// TIA Portal V20 export
// export: Created 2025-12-01T14:57:27.8084836Z, ExportSetting None, DisplayName Totally Integrated Automation Portal, DisplayVersion V20 Update 3, DisplayName TIA Portal Openness, DisplayVersion V20 Update 3, DisplayName TIA Portal Version Control Interface, DisplayVersion V20 Update 3, DisplayName STEP 7 Professional, DisplayVersion V20 Update 3, DisplayName STEP 7 Safety, DisplayVersion V20 Update 2, DisplayName WinCC Basic/Comfort/Advanced, DisplayVersion V20 Update 3, DisplayName WinCC Professional, DisplayVersion V20 Update 3, DisplayName WinCC Unified, DisplayVersion V20 Update 3
FUNCTION_BLOCK "FB603_EntradaMovil_Frontal_Quimarox"   // FB603, LAD
{ S7_Optimized_Access := 'FALSE' }
// stored: AutoNumber false, SetENOAutomatically false
   VAR_INPUT
      MesaDeCarga : UInt;
      ID_Quimarox : UInt;
      ID_Elemento : UInt;
      EnTension : Bool;
      Termico_Tilt : Bool;
      pHs_PosicionCarga : Bool;
      pHs_Protrusion : Bool;
      En_PosicionReposo : Bool;
      Corte_PosicionReposo : Bool;
      Corte_PosicionCarga : Bool;
      En_PosicionCarga : Bool;
      PRV_AVTF : Bool;
      PRV_DescargaActiva : Bool;
      V_FILTRO_pHsPresencia : Int;
      Pto_Ajuste_1 : Int;
      Pto_Ajuste_2 : Int;
      Pto_Ajuste_3 : Int;
      Pto_Ajuste_4 : Int;
      Pto_Ajuste_5 : Int;
      Pto_Ajuste_6 : Int;
   END_VAR
   VAR_OUTPUT
      Permiso_DeCarga : Bool;
      PararElevador : Bool;
      ElevadorEnLenta : Bool;
      AvanceCorreas : Bool;
      Ir_PosicionReposo : Bool;
      Ir_PosicionCarga : Bool;
   END_VAR
   VAR_IN_OUT
      ROUTING_Destino : UInt;
      ROUTING_Etiqueta : UDInt;
   END_VAR
   VAR
      TMP_EnTension { S7_SetPoint := 'True'} : "FB910_CNT_UHS";
      FILTRO_pHsPresencia { S7_SetPoint := 'True'} : "FB910_CNT_UHS";
      EstadoAsociadoEnMesa : UInt;
      Aux_PeineDeCarga : UInt;
   END_VAR
   VAR_TEMP
      MesaQuimarox : UInt;
      PeineReservado : UInt;
      TMP_PeineLiberar : UInt;
      NumeroUT : UInt;
      EsMesaTL : Bool;
      FILTRO_PosicionCarga : Bool;
   END_VAR
BEGIN

NETWORK
TITLE = ERROR - Rearme
/////////////////////////////////////////////////////////////
/////////////////////////////////////////////////////////////
/////////////////////////////////////////////////////////////
// Rearne de Errores
      SET;
      A     "DB902_Estado_ZonaMesa".EstadoMesas[#MesaDeCarga].Rearme_CBx;
      O     "DB902_Estado_ZonaMesa".EstadoMesas[#MesaDeCarga].PerReset_CBx;
      R     "DB900_Estado_Mesas".EstadoVI[#MesaDeCarga].Error_Mx;
      R     "DB900_Estado_Mesas".EstadoVI[#MesaDeCarga].Err_Protusion;
      R     "DB900_Estado_Mesas".EstadoVI[#MesaDeCarga].Err_TOut_Avance_E1_E3;
      R     "DB900_Estado_Mesas".EstadoVI[#MesaDeCarga].Err_Tout_Sacar;
      R     "DB900_Estado_Mesas".EstadoVI[#MesaDeCarga].Err_Tout_Recoger;
      R     "DB900_Estado_Mesas".EstadoVI[#MesaDeCarga].Err_DatosPLC;
      R     "DB900_Estado_Mesas".EstadoVI[#MesaDeCarga].Err_Termico_E2_E4;



NETWORK
TITLE = HMI - Manual
/////////////////////////////////////////////////////////////
/////////////////////////////////////////////////////////////
/////////////////////////////////////////////////////////////
// Para HMI >>> Manual
      SET;
      O     "DB902_Estado_ZonaMesa".EstadoMesas[#MesaDeCarga].Manual_CBx;
      =     "DB900_Estado_Mesas".EstadoVI[#MesaDeCarga].Manual;



NETWORK
TITLE = HMI - Entradas y Salidas de la Mesa
/////////////////////////////////////////////////////////////
/////////////////////////////////////////////////////////////
/////////////////////////////////////////////////////////////
// Entradas
      SET;
      A     #pHs_PosicionCarga;
      =     "DB900_Estado_Mesas".EstadoVI[#MesaDeCarga].En_PHS_1;
      SET;
      A     #pHs_Protrusion;
      =     "DB900_Estado_Mesas".EstadoVI[#MesaDeCarga].En_pHs_Prot1;

      SET;  // Solo el TILT
      A     #Termico_Tilt;
      =     "DB900_Estado_Mesas".EstadoVI[#MesaDeCarga].En_Termico2;

      SET;
      A     #En_PosicionReposo;
      =     "DB904_Estado_Maquinas".EstadoVI[#MesaDeCarga].Byte8_bit4;
      SET;
      A     #Corte_PosicionReposo;
      =     "DB904_Estado_Maquinas".EstadoVI[#MesaDeCarga].Byte7_bit6;
      SET;
      A     #Corte_PosicionCarga;
      =     "DB904_Estado_Maquinas".EstadoVI[#MesaDeCarga].Byte7_bit7;
      SET;
      A     #En_PosicionCarga;
      =     "DB904_Estado_Maquinas".EstadoVI[#MesaDeCarga].Byte8_bit5;


// Salidas
      SET;
      A     #Permiso_DeCarga;
      =     "DB900_Estado_Mesas".EstadoVI[#MesaDeCarga].Sa_Extender_Empujador;
      SET;
      A     #Ir_PosicionReposo;
      =     "DB900_Estado_Mesas".EstadoVI[#MesaDeCarga].Sa_Trans_Baj;
      SET;
      A     #Ir_PosicionCarga;
      =     "DB900_Estado_Mesas".EstadoVI[#MesaDeCarga].Sa_Trans_Sub;



NETWORK
TITLE = Comprobacion de que la MESA es de TRACKING
/////////////////////////////////////////////////////////////////////////////////////
/////////////////////////////////////////////////////////////////////////////////////
/////////////////////////////////////////////////////////////////////////////////////
// Comprobar si es una Mesa de Tracking o Routing
      SET;
      A     "DB850_DefinicionMesas".Mesa[#MesaDeCarga].ConfigMesa.MesaTL;
      =     #EsMesaTL;



REGION Network 5: TMP - Espera En Tension
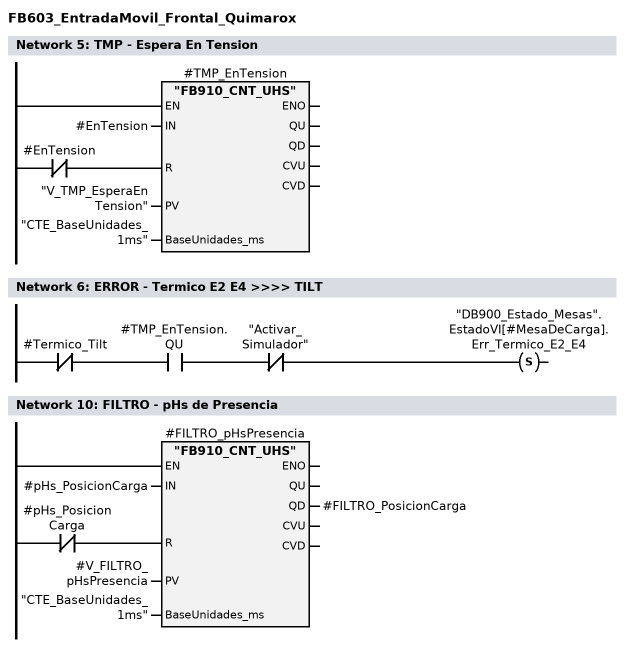
   RUNG wire#powerrail
      #TMP_EnTension(R := wire#w1, IN := #EnTension, PV := "V_TMP_EsperaEnTension", BaseUnidades_ms := "CTE_BaseUnidades_1ms", QU =>, QD =>, CVU =>, CVD =>)
   END_RUNG
   RUNG wire#powerrail
      I_Contact( #EnTension )
   END_RUNG wire#w1
   // the same network as SCL:
   #TMP_EnTension(IN := #EnTension,   // "FB910_CNT_UHS"
                  R := NOT #EnTension,
                  PV := "V_TMP_EsperaEnTension",
                  BaseUnidades_ms := "CTE_BaseUnidades_1ms");
END_REGION

REGION Network 6: ERROR - Termico E2 E4 >>>> TILT
   RUNG wire#powerrail
      I_Contact( #Termico_Tilt )
      Contact( #TMP_EnTension.QU )
      I_Contact( "Activar_Simulador" )
      S_Coil( "DB900_Estado_Mesas".EstadoVI[#MesaDeCarga].Err_Termico_E2_E4 )
   END_RUNG
   // the same network as SCL:
   IF NOT #Termico_Tilt AND #TMP_EnTension.QU AND NOT "Activar_Simulador" THEN
       "DB900_Estado_Mesas".EstadoVI[#MesaDeCarga].Err_Termico_E2_E4 := TRUE;
   END_IF;
END_REGION

NETWORK
TITLE = INICIALIZACION - Previa
/////////////////////////////////////////////////////////////////////////////////////
/////////////////////////////////////////////////////////////////////////////////////
/////////////////////////////////////////////////////////////////////////////////////
      CLR;
      =     #PararElevador;
      =     #ElevadorEnLenta;

      CLR;
      =     #Permiso_DeCarga;

      CLR;
      =     #AvanceCorreas;
      =     #Ir_PosicionReposo;
      =     #Ir_PosicionCarga;



NETWORK
TITLE = SISTEMA - Reset
/////////////////////////////////////////////////////////////
/////////////////////////////////////////////////////////////
/////////////////////////////////////////////////////////////
// - Existe RESET ??
      SET;
      AN    "DB902_Estado_ZonaMesa".EstadoMesas[#MesaDeCarga].PerReset_CBx;  //#Estado_CBx.PerReset_CBx
      JC    NoRealizandose_Reset;

      L     0;
      T     #EstadoAsociadoEnMesa;


/////////////////////////////////////////////////////////////
/////////////////////////////////////////////////////////////
/////////////////////////////////////////////////////////////
// - Final Tratamiento del RESET
NoRealizandose_Reset:NOP   0;



NETWORK
TITLE = >>>>>>>>>>>>>>>>>>>>>>>>>>>>>>>>>>>>>>>>>>>>>>>>>>>>>>>>>>>>>>>>>>>

REGION Network 10: FILTRO - pHs de Presencia
   RUNG wire#powerrail
      #FILTRO_pHsPresencia(R := wire#w1, IN := #pHs_PosicionCarga, PV := #V_FILTRO_pHsPresencia, BaseUnidades_ms := "CTE_BaseUnidades_1ms", QU =>, QD => #FILTRO_PosicionCarga, CVU =>, CVD =>)
   END_RUNG
   RUNG wire#powerrail
      I_Contact( #pHs_PosicionCarga )
   END_RUNG wire#w1
   // the same network as SCL:
   #FILTRO_pHsPresencia(IN := #pHs_PosicionCarga,   // "FB910_CNT_UHS"
                        R := NOT #pHs_PosicionCarga,
                        PV := #V_FILTRO_pHsPresencia,
                        BaseUnidades_ms := "CTE_BaseUnidades_1ms",
                        QD => #FILTRO_PosicionCarga);
END_REGION

NETWORK
TITLE = >>>>>>>>>>>>>>>>>>>>>>>>>>>>>>>>>>>>>>>>>>>>>>>>>>>>>>>>>>>>>>>>>>>

NETWORK
TITLE = Disrtibucion >>> Control Etapa Activa
/////////////////////////////////////////////////////////////////////////////////////
/////////////////////////////////////////////////////////////////////////////////////
/////////////////////////////////////////////////////////////////////////////////////
// listado de saltos de programa
      L     #EstadoAsociadoEnMesa;
      JL    ESTADO_PorDefecto;

      JU    ETAPA_00_EnReset;
      JU    ETAPA_01_EnReposo;

      JU    ETAPA_02_PrevioCarga_ComprobarRuta;
      JU    ETAPA_03_PrevioCarga_ReservaPeine;
      JU    ETAPA_04_PrevioCarga_Sincroniza;
      JU    ETAPA_05_PrevioCarga_MoverPosicionDeCarga;
      JU    ETAPA_06_CargaDelPeine;
      JU    ETAPA_07_FinCargaDelPeine;
      JU    ETAPA_08_VolverReposo;

      JU    ESTADO_PorDefecto;

      JU    ETAPA_10_ResetCargado_ComprobarRuta;
      JU    ETAPA_11_ResetVacio_MoverPosicionDeReposo;

ESTADO_PorDefecto:JU    FinFuncion;



NETWORK
TITLE = ETAPA 00 >>> Etapa Reset >>>> PENDIENTE
/////////////////////////////////////////////////////////////////////////////////////
/////////////////////////////////////////////////////////////////////////////////////
/////////////////////////////////////////////////////////////////////////////////////
ETAPA_00_EnReset:NOP   0;
      SET;
      =     "DB900_Estado_Mesas".EstadoVI[#MesaDeCarga].Etapas_Reset;

/////////////////////////////////////////////////////////////////////////////////////
// error de protusion
      SET;
      AN    #pHs_Protrusion;
      JC    ErrorProtrusion;


/////////////////////////////////////////////////////////////////////////////////////
// Tiene que estar en Marcha y Sin Error para continuar
      SET;
      AN    "DB902_Estado_ZonaMesa".EstadoMesas[#MesaDeCarga].Marcha_CBx;
      O     "DB902_Estado_ZonaMesa".EstadoMesas[#MesaDeCarga].Error_CBx;
      JC    ET00_PararElevador;



/////////////////////////////////////////////////////////////////////////////////////
// En Resposo
      SET;
      A     #En_PosicionReposo;
      JC    ET00_IrEtapa_01_EnReposo;

/////////////////////////////////////////////////////////////////////////////////////
// NO Reposo - Vacio
      SET;
      AN    #FILTRO_PosicionCarga;
      JC    ET00_IrEtapa_11_ResetVacio_MoverPosicionReposo;

/////////////////////////////////////////////////////////////////////////////////////
// NO Reposo - Con Carga
      SET;
      A     #FILTRO_PosicionCarga;
      JC    ET00_IrEtapa_10_ResetCargado_ComprobarRuta;


/////////////////////////////////////////////////////////////////////////////////////
// Final del Reparto  ?????? No DEBE LLEGAR AQUI
      BE;


/////////////////////////////////////////////////////////////////////////////////////
/////////////////////////////////////////////////////////////////////////////////////
/////////////////////////////////////////////////////////////////////////////////////
ET00_PararElevador:NOP   0;
      SET;
      =     #PararElevador;
      BE;


/////////////////////////////////////////////////////////////////////////////////////
/////////////////////////////////////////////////////////////////////////////////////
/////////////////////////////////////////////////////////////////////////////////////
ET00_IrEtapa_01_EnReposo:NOP   0;
      L     1;
      T     #EstadoAsociadoEnMesa;
      JU    ETAPA_01_EnReposo;

/////////////////////////////////////////////////////////////////////////////////////
ET00_IrEtapa_10_ResetCargado_ComprobarRuta:NOP   0;
      L     10;
      T     #EstadoAsociadoEnMesa;
      JU    ETAPA_10_ResetCargado_ComprobarRuta;

/////////////////////////////////////////////////////////////////////////////////////
ET00_IrEtapa_11_ResetVacio_MoverPosicionReposo:NOP   0;
      L     11;
      T     #EstadoAsociadoEnMesa;
      JU    ETAPA_11_ResetVacio_MoverPosicionDeReposo;



NETWORK
TITLE = ETAPA 01 >>> Etapa Reposo >>> Esta Vacia
/////////////////////////////////////////////////////////////////////////////////////
/////////////////////////////////////////////////////////////////////////////////////
/////////////////////////////////////////////////////////////////////////////////////
// estado reposo
ETAPA_01_EnReposo:NOP   0;
      SET;
      =     "DB900_Estado_Mesas".EstadoVI[#MesaDeCarga].Etapa_Vacia;


/////////////////////////////////////////////////////////////////////////////////////
// error de protusion
      SET;
      AN    #pHs_Protrusion;
      JC    ErrorProtrusion;

/////////////////////////////////////////////////////////////////////////////////////
/////////////////////////////////////////////////////////////////////////////////////
/////////////////////////////////////////////////////////////////////////////////////
// Si Viene un Peine >>> Reservado para el Elemento >>> LIBERAR Peine
      SET;  // --- Sin Ventana
      AN    "DB602_ElementosQuimarox".Quimarox[#ID_Quimarox].Elementos[#ID_Elemento].Hay_Carrier_en_ventana;
      JC    ET01_PorReserva_NoLiberarPeine;

      L     "DB602_ElementosQuimarox".Quimarox[#ID_Quimarox].Elementos[#ID_Elemento].Numero_carrier;
      T     #TMP_PeineLiberar;

      SET;  // --- Sin Reserva
      AN    "DB601_PeinesQuimarox".Quimarox[#ID_Quimarox].vagon[#TMP_PeineLiberar].vagon_reservado_carga;
      JC    ET01_PorReserva_NoLiberarPeine;

      SET;  // --- No es para el elemento
      L     "DB601_PeinesQuimarox".Quimarox[#ID_Quimarox].vagon[#TMP_PeineLiberar].punto_entrada_carga;
      L     #ID_Elemento;
      <>I;
      JC    ET01_PorReserva_NoLiberarPeine;

/////////////////////////////////////////////////////////////////////////////////////
      SET;  // --- Liberar Peine
      R     "DB601_PeinesQuimarox".Quimarox[#ID_Quimarox].vagon[#TMP_PeineLiberar].vagon_reservado_carga;

      L     0;
      T     "DB601_PeinesQuimarox".Quimarox[#ID_Quimarox].vagon[#TMP_PeineLiberar].punto_entrada_carga;

/////////////////////////////////////////////////////////////////////////////////////
ET01_PorReserva_NoLiberarPeine:NOP   0;


/////////////////////////////////////////////////////////////////////////////////////
/////////////////////////////////////////////////////////////////////////////////////
/////////////////////////////////////////////////////////////////////////////////////
// Esta poscionado Correctamente
      SET;
      AN    #PRV_AVTF;
      AN    #FILTRO_PosicionCarga;
      A     #pHs_Protrusion;
      AN    #En_PosicionReposo;
      JC    ET01_IrEtapa_08_VolverReposo;

/////////////////////////////////////////////////////////////////////////////////////
      SET;
      AN    #PRV_AVTF;
      AN    #FILTRO_PosicionCarga;
      A     #pHs_Protrusion;
      JC    FinFuncion;

/////////////////////////////////////////////////////////////////////////////////////
      SET;
      A     #PRV_AVTF;
      AN    #FILTRO_PosicionCarga;
      A     #pHs_Protrusion;
      JC    ET01_IrEtapa_02_PrevioCarga_ComprobarRuta;

      BE;


/////////////////////////////////////////////////////////////////////////////////////
ET01_IrEtapa_08_VolverReposo:NOP   0;
      L     8;
      T     #EstadoAsociadoEnMesa;
      JU    ETAPA_08_VolverReposo;

/////////////////////////////////////////////////////////////////////////////////////
ET01_IrEtapa_02_PrevioCarga_ComprobarRuta:NOP   0;
      L     2;
      T     #EstadoAsociadoEnMesa;
      JU    ETAPA_02_PrevioCarga_ComprobarRuta;



NETWORK
TITLE = ETAPA 02 >>> Comprobar Ruta >>>>> OJO!!!!!!!!!!!!!!!
/////////////////////////////////////////////////////////////////////////////////////
// estado preparar carga
ETAPA_02_PrevioCarga_ComprobarRuta:NOP   0;
      SET;
      =     "DB900_Estado_Mesas".EstadoVI[#MesaDeCarga].Etapa_Vacia;

/////////////////////////////////////////////////////////////////////////////////////
// Error de Protrusion
      SET;
      AN    #pHs_Protrusion;
      JC    ErrorProtrusion;

/////////////////////////////////////////////////////////////////////////////////////
/// --- Comprobacion del TIPO de MESA
      SET;
      AN    #EsMesaTL;
      JC    TRACKING_ComprobarRuta;
      JU    ROUTING_ComprobarRuta;

/////////////////////////////////////////////////////////////////////////////////////
/////////////////////////////////////////////////////////////////////////////////////
/////////////////////////////////////////////////////////////////////////////////////
/// --- Comprobacion de Ruta en una MESA de ROUTING
ROUTING_ComprobarRuta:NOP   0;
      L     #ROUTING_Destino;
      L     0;
      ==I;
      JC    FinFuncion;
      JU    FINAL_ComprobacionDeRuta;

/////////////////////////////////////////////////////////////////////////////////////
/////////////////////////////////////////////////////////////////////////////////////
/////////////////////////////////////////////////////////////////////////////////////
/// --- Comprobacion de Ruta en una MESA de TRACKING
TRACKING_ComprobarRuta:NOP   0;
      L     "DB810_ColasMesas".Colas[#MesaDeCarga].UT_PrimeraMesa;
      T     #NumeroUT;

      SET;
      L     #NumeroUT;  // Debe existir UT
      L     0;
      ==I;
      JC    FinFuncion;

// si la mesa actual es la de destino, es que aun no tiene ruta, y tenemos que esperar
      SET;
      L     "DB812_UTs_Control".UT[#NumeroUT].MesaActual;
      L     "DB812_UTs_Control".UT[#NumeroUT].MesaDestino;
      ==I;
      JC    FinFuncion;

      SET;
      L     0;
      L     "DB812_UTs_Control".UT[#NumeroUT].MesaDestino;
      ==I;
      JC    FinFuncion;

      JU    FINAL_ComprobacionDeRuta;

/////////////////////////////////////////////////////////////////////////////////////
/////////////////////////////////////////////////////////////////////////////////////
/////////////////////////////////////////////////////////////////////////////////////
/// --- Final de la Comprobacion de Ruta
//      si tenemos destino, pasamos a reservar peine de carga
FINAL_ComprobacionDeRuta:NOP   0;
      L     3;
      T     #EstadoAsociadoEnMesa;
      JU    ETAPA_03_PrevioCarga_ReservaPeine;  // si ya hemos extraido la orden, pasamos a extraer el destino



NETWORK
TITLE = ETAPA 03 >>> Reserva Peine
/////////////////////////////////////////////////////////////////////////////////////
/////////////////////////////////////////////////////////////////////////////////////
/////////////////////////////////////////////////////////////////////////////////////
// extracción destino y reserva de peine
ETAPA_03_PrevioCarga_ReservaPeine:NOP   0;
      SET;
      =     "DB900_Estado_Mesas".EstadoVI[#MesaDeCarga].Etapa_Vacia;


/////////////////////////////////////////////////////////////////////////////////////
      SET;
      AN    #pHs_Protrusion;
      JC    ErrorProtrusion;

/////////////////////////////////////////////////////////////////////////////////////
// rearme del error si ha desaparecido la caja   OJO!!!!!!!CAMBIADO
      SET;
      AN    #PRV_AVTF;
      AN    #FILTRO_PosicionCarga;
      A     #pHs_Protrusion;
      A     "DB902_Estado_ZonaMesa".EstadoMesas[#MesaDeCarga].Rearme_CBx;
      JC    ET03_IrEtapa_01_EnReposo;


/////////////////////////////////////////////////////////////////////////////////////
/////////////////////////////////////////////////////////////////////////////////////
/////////////////////////////////////////////////////////////////////////////////////
// reserva de peine >>> Mesa Movil Frontal (3)
      CALL  "FC602_ReservaPeine"
      ( ID_Quimarox          := #ID_Quimarox,
        ID_ElementoPeticion  := #ID_Elemento,
        TipoDeElemento       := 3,
        NumeroPeineReservado := #PeineReservado
      );

      SET;
      L     #PeineReservado;
      L     0;
      ==I;
      JC    FinFuncion;

/////////////////////////////////////////////////////////////////////////////////////
/////////////////////////////////////////////////////////////////////////////////////
/////////////////////////////////////////////////////////////////////////////////////
      L     #PeineReservado;  // recogemos la peticion
      T     #Aux_PeineDeCarga;

      L     4;
      T     #EstadoAsociadoEnMesa;
      JU    ETAPA_04_PrevioCarga_Sincroniza;


/////////////////////////////////////////////////////////////////////////////////////
ET03_IrEtapa_01_EnReposo:NOP   0;
      L     1;
      T     #EstadoAsociadoEnMesa;
      JU    ETAPA_01_EnReposo;



NETWORK
TITLE = ETAPA 04 >>> Sincronizacion
/////////////////////////////////////////////////////////////////////////////////////
/////////////////////////////////////////////////////////////////////////////////////
/////////////////////////////////////////////////////////////////////////////////////
// a la espera de la sincronización con el peine reservado para nosotros
ETAPA_04_PrevioCarga_Sincroniza:NOP   0;
      SET;
      =     "DB900_Estado_Mesas".EstadoVI[#MesaDeCarga].Etapas_Carga_E1;


/////////////////////////////////////////////////////////////////////////////////////
// Error de Protrusion
      SET;
      AN    #pHs_Protrusion;
      JC    ErrorProtrusion;

/////////////////////////////////////////////////////////////////////////////////////
// ahora que ya estamos los datos de nuestro elemento comprobamos lo siguiente
// que tenemos delante el carrier que tenemos reservado para la carga
// que el carrier reservado para la carga está en ventana
      SET;
      A     "DB602_ElementosQuimarox".Quimarox[#ID_Quimarox].Elementos[#ID_Elemento].Hay_Carrier_en_ventana;
      A(;
      L     "DB602_ElementosQuimarox".Quimarox[#ID_Quimarox].Elementos[#ID_Elemento].Numero_carrier;  //#datos_elemento.Numero_carrier
      L     #Aux_PeineDeCarga;
      ==I;
      );
      JC    ET04_IrEtapa_05_MoverPosicionDeCarga;

      BE;

/////////////////////////////////////////////////////////////////////////////////////
ET04_IrEtapa_05_MoverPosicionDeCarga:NOP   0;
      L     5;  // saltamos al inicio de posicionamiento para carga
      T     #EstadoAsociadoEnMesa;
      JU    ETAPA_05_PrevioCarga_MoverPosicionDeCarga;



NETWORK
TITLE = ETAPA 05 >>> Mover Posicion de Carga
/////////////////////////////////////////////////////////////////////////////////////
/////////////////////////////////////////////////////////////////////////////////////
/////////////////////////////////////////////////////////////////////////////////////
ETAPA_05_PrevioCarga_MoverPosicionDeCarga:NOP   0;
      SET;
      =     "DB900_Estado_Mesas".EstadoVI[#MesaDeCarga].Etapas_Carga_E1;


      SET;
      A     #En_PosicionCarga;
      JC    ET05_IrEtapa_06_CargaDelPeine;

      SET;
      =     #Ir_PosicionCarga;
      =     #AvanceCorreas;
      =     #Permiso_DeCarga;
      CLR;
      =     #Ir_PosicionReposo;


/////////////////////////////////////////////////////////////////////////////////////
// como estamos metiendo el transportador, tenemos que vigilar que no tarda demasiado en entrar
      L     "DB602_ElementosQuimarox".Quimarox[#ID_Quimarox].Elementos[#ID_Elemento].Avance_carrier;
      L     #Pto_Ajuste_1;
      <=I;
      JC    ET05_VelocidadNormal;

      SET;
      =     #ElevadorEnLenta;

/////////////////////////////////////////////////////////////////////////////////////
      L     "DB602_ElementosQuimarox".Quimarox[#ID_Quimarox].Elementos[#ID_Elemento].Avance_carrier;
      L     #Pto_Ajuste_2;
      >=I;
      JC    ErrorMoverPosicionCarga;  // error de movimiento al sacar el transportador

      BE;


/////////////////////////////////////////////////////////////////////////////////////
ET05_VelocidadNormal:CLR;
      =     #ElevadorEnLenta;
      BE;

/////////////////////////////////////////////////////////////////////////////////////
ET05_IrEtapa_06_CargaDelPeine:NOP   0;
      CLR;
      =     #Ir_PosicionCarga;
      =     #AvanceCorreas;

      L     6;
      T     #EstadoAsociadoEnMesa;
      JU    ETAPA_06_CargaDelPeine;



NETWORK
TITLE = ETAPA 06 >>> Carga En Peine
/////////////////////////////////////////////////////////////////////////////////////
/////////////////////////////////////////////////////////////////////////////////////
/////////////////////////////////////////////////////////////////////////////////////
ETAPA_06_CargaDelPeine:NOP   0;
      SET;
      =     "DB900_Estado_Mesas".EstadoVI[#MesaDeCarga].Etapas_Carga_E1;


      SET;
      =     #Permiso_DeCarga;

/////////////////////////////////////////////////////////////////////////////////////
      SET;  // hemos cargado correctamente y generamos los datos para el peine
      A     #FILTRO_PosicionCarga;
      AN    #PRV_AVTF;
      A     #pHs_Protrusion;
      JC    ET06_IrEtapa_07_FinCargaDelPeine;

/////////////////////////////////////////////////////////////////////////////////////
// aqui tenemos que vigilar que nos se nos está cerrado la ventana intentando cargar
// primero comprobamos que no tenemos ya la ventana cerrada, porque sino tenemos que parar el elevador
      SET;
      AN    "DB602_ElementosQuimarox".Quimarox[#ID_Quimarox].Elementos[#ID_Elemento].Hay_Carrier_en_ventana;
      A(;
      ON    #pHs_Protrusion;
      O     #FILTRO_PosicionCarga;
      );
      JC    ErrorCargaDelPeine;

/////////////////////////////////////////////////////////////////////////////////////
      SET;
      AN    "DB602_ElementosQuimarox".Quimarox[#ID_Quimarox].Elementos[#ID_Elemento].Hay_Carrier_en_ventana;
      AN    #FILTRO_PosicionCarga;
      A     #pHs_Protrusion;
      AN    #PRV_AVTF;
      JC    ET06_PasadoVagon_SinCargar;

/////////////////////////////////////////////////////////////////////////////////////
// Deberia Haber Cargado en este punto
      SET;
      A     "DB602_ElementosQuimarox".Quimarox[#ID_Quimarox].Elementos[#ID_Elemento].Hay_Carrier_en_ventana;
      A(;
      L     "DB602_ElementosQuimarox".Quimarox[#ID_Quimarox].Elementos[#ID_Elemento].Avance_carrier;
      L     #Pto_Ajuste_3;
      >=I;
      );
      AN    #pHs_Protrusion;
      JC    ErrorProtrusion;

/////////////////////////////////////////////////////////////////////////////////////
      SET;
      A     "DB602_ElementosQuimarox".Quimarox[#ID_Quimarox].Elementos[#ID_Elemento].Hay_Carrier_en_ventana;
      AN    #FILTRO_PosicionCarga;
      A(;
      L     "DB602_ElementosQuimarox".Quimarox[#ID_Quimarox].Elementos[#ID_Elemento].Avance_carrier;
      L     #Pto_Ajuste_3;
      >=I;
      );
      JC    ErrorCargaDelPeine;

/////////////////////////////////////////////////////////////////////////////////////
      SET;
      A     "DB602_ElementosQuimarox".Quimarox[#ID_Quimarox].Elementos[#ID_Elemento].Hay_Carrier_en_ventana;
      A(;
      L     "DB602_ElementosQuimarox".Quimarox[#ID_Quimarox].Elementos[#ID_Elemento].Avance_carrier;
      L     #Pto_Ajuste_3;
      >=I;
      );
      A     #PRV_AVTF;
      JC    ErrorCargaDelPeine;

      BE;


/////////////////////////////////////////////////////////////////////////////////////
ET06_PasadoVagon_SinCargar:NOP   0;
      CLR;
      =     #ElevadorEnLenta;
      =     #Permiso_DeCarga;

      CLR;
      =     "DB601_PeinesQuimarox".Quimarox[#ID_Quimarox].vagon[#Aux_PeineDeCarga].vagon_reservado_carga;  //#datos_peine_tmp.vagon_reservado_carga
      L     0;
      T     "DB601_PeinesQuimarox".Quimarox[#ID_Quimarox].vagon[#Aux_PeineDeCarga].punto_entrada_carga;
      T     #Aux_PeineDeCarga;

      L     8;
      T     #EstadoAsociadoEnMesa;
      JU    ETAPA_08_VolverReposo;

/////////////////////////////////////////////////////////////////////////////////////
ET06_ElevadorNormal:CLR;
      =     #ElevadorEnLenta;
      BE;

/////////////////////////////////////////////////////////////////////////////////////
ET06_IrEtapa_07_FinCargaDelPeine:NOP   0;
      L     7;
      T     #EstadoAsociadoEnMesa;
      JU    ETAPA_07_FinCargaDelPeine;



NETWORK
TITLE = ETAPA 07 >>> Fin de Carga >>> Paso de Datos al VAGON >>>>> OJO!!!!!!!!!!!!!!!
/////////////////////////////////////////////////////////////////////////////////////
/////////////////////////////////////////////////////////////////////////////////////
/////////////////////////////////////////////////////////////////////////////////////
ETAPA_07_FinCargaDelPeine:NOP   0;
      SET;
      =     "DB900_Estado_Mesas".EstadoVI[#MesaDeCarga].Etapas_Descarga_S0;

      SET;
      =     #Permiso_DeCarga;

/////////////////////////////////////////////////////////////////////////////////////
// Error de Protusion
      SET;
      AN    #pHs_Protrusion;
      JC    ErrorProtrusion;


/////////////////////////////////////////////////////////////////////////////////////
//// Cargado Correctamente
      SET;
      AN    #FILTRO_PosicionCarga;
      A     #pHs_Protrusion;
      JC    FINALIZADO_CargaDelPeine;

      BE;


/////////////////////////////////////////////////////////////////////////////////////
/////////////////////////////////////////////////////////////////////////////////////
/////////////////////////////////////////////////////////////////////////////////////
// cargamos los datos de la UT al peine   >>>>> DEPENDIENDO DE TIPO DE DATOS
FINALIZADO_CargaDelPeine:NOP   0;
      SET;
      =     "DB601_PeinesQuimarox".Quimarox[#ID_Quimarox].vagon[#Aux_PeineDeCarga].Carrier_Cargado;

      SET;
      AN    #EsMesaTL;
      JC    TRACKING_PasoDeDatos;
      JU    ROUTING_PasoDeDatos;

/////////////////////////////////////////////////////////////////////////////////////
// --- DATOS DE ROUTING
ROUTING_PasoDeDatos:NOP   0;
      L     0;
      T     "DB601_PeinesQuimarox".Quimarox[#ID_Quimarox].vagon[#Aux_PeineDeCarga].DatosCarga.Mckey;
      L     #MesaDeCarga;
      T     "DB601_PeinesQuimarox".Quimarox[#ID_Quimarox].vagon[#Aux_PeineDeCarga].DatosCarga.MesaOrigen;
      L     #ROUTING_Destino;
      T     "DB601_PeinesQuimarox".Quimarox[#ID_Quimarox].vagon[#Aux_PeineDeCarga].DatosCarga.MesaDestino;
      T     "DB601_PeinesQuimarox".Quimarox[#ID_Quimarox].vagon[#Aux_PeineDeCarga].Destino_principal;

      L     #ROUTING_Etiqueta;
      T     "DB601_PeinesQuimarox".Quimarox[#ID_Quimarox].vagon[#Aux_PeineDeCarga].DatosCarga.EtiquetaRouter;

      L     "CTE_Evento_QCAR";
      T     "DB601_PeinesQuimarox".Quimarox[#ID_Quimarox].vagon[#Aux_PeineDeCarga].EventoAGenerar;

      L     0;
      T     #ROUTING_Destino;
      T     #ROUTING_Etiqueta;

      JU    FINAL_PasoDeDatos;

/////////////////////////////////////////////////////////////////////////////////////
// --- DATOS DE TRACKING
TRACKING_PasoDeDatos:NOP   0;
      L     "DB810_ColasMesas".Colas[#MesaDeCarga].UT_PrimeraMesa;
      T     #NumeroUT;

      L     "DB812_UTs_Control".UT[#NumeroUT].Mckey;
      T     "DB601_PeinesQuimarox".Quimarox[#ID_Quimarox].vagon[#Aux_PeineDeCarga].DatosCarga.Mckey;
      L     "DB812_UTs_Control".UT[#NumeroUT].MesaActual;
      T     "DB601_PeinesQuimarox".Quimarox[#ID_Quimarox].vagon[#Aux_PeineDeCarga].DatosCarga.MesaOrigen;
      L     "DB812_UTs_Control".UT[#NumeroUT].MesaDestino;
      T     "DB601_PeinesQuimarox".Quimarox[#ID_Quimarox].vagon[#Aux_PeineDeCarga].DatosCarga.MesaDestino;
      T     "DB601_PeinesQuimarox".Quimarox[#ID_Quimarox].vagon[#Aux_PeineDeCarga].Destino_principal;

      L     "DB814_UTs_Etiqueta".UT[#NumeroUT].EtiquetaRouter;
      T     "DB601_PeinesQuimarox".Quimarox[#ID_Quimarox].vagon[#Aux_PeineDeCarga].DatosCarga.EtiquetaRouter;

      L     "CTE_Evento_QCAR";
      T     "DB601_PeinesQuimarox".Quimarox[#ID_Quimarox].vagon[#Aux_PeineDeCarga].EventoAGenerar;
      L     131;
      T     "DB812_UTs_Control".UT[#NumeroUT].EstadoEventoAGenerar;

// Borrar UT Sin Avisar al JDT >>>> OJO
      CALL  "FC722_EliminarUT_DeMesa"
      ( NumeroUT := #NumeroUT
      );


/////////////////////////////////////////////////////////////////////////////////////
/////////////////////////////////////////////////////////////////////////////////////
/////////////////////////////////////////////////////////////////////////////////////
FINAL_PasoDeDatos:NOP   0;
      CLR;
      =     #ElevadorEnLenta;
      =     #Permiso_DeCarga;

      CLR;
      =     "DB601_PeinesQuimarox".Quimarox[#ID_Quimarox].vagon[#Aux_PeineDeCarga].vagon_reservado_carga;  //#datos_peine_tmp.vagon_reservado_carga

      L     0;
      T     "DB601_PeinesQuimarox".Quimarox[#ID_Quimarox].vagon[#Aux_PeineDeCarga].punto_entrada_carga;
      T     #Aux_PeineDeCarga;

// pasamos a la etapa de volver a posicion de reposo
      L     8;
      T     #EstadoAsociadoEnMesa;
      JU    ETAPA_08_VolverReposo;



NETWORK
TITLE = ETAPA 08 >>> Volver a Posicion de Reposo
/////////////////////////////////////////////////////////////////////////////////////
/////////////////////////////////////////////////////////////////////////////////////
/////////////////////////////////////////////////////////////////////////////////////
ETAPA_08_VolverReposo:NOP   0;
      SET;
      =     "DB900_Estado_Mesas".EstadoVI[#MesaDeCarga].Etapas_Descarga_S0;

      SET;
      A     #En_PosicionReposo;
      JC    ET08_IrEtapa_01_Vacia;

/////////////////////////////////////////////////////////////////////////////////////
// No pasar a Reposo Hasta pasar este punto
      SET;
      L     "DB602_ElementosQuimarox".Quimarox[#ID_Quimarox].Elementos[#ID_Elemento].Avance_carrier;  //#datos_elemento.Avance_carrier
      L     #Pto_Ajuste_4;
      <=I;
      JC    FinFuncion;

      SET;
      =     #Ir_PosicionReposo;


/////////////////////////////////////////////////////////////////////////////////////
/////////////////////////////////////////////////////////////////////////////////////
/////////////////////////////////////////////////////////////////////////////////////
      SET;
      L     "DB602_ElementosQuimarox".Quimarox[#ID_Quimarox].Elementos[#ID_Elemento].Avance_carrier;  //#datos_elemento.Avance_carrier
      L     #Pto_Ajuste_5;
      <=I;
      JC    ET05_VelocidadNormal;

      SET;
      =     #ElevadorEnLenta;

/////////////////////////////////////////////////////////////////////////////////////
// error de movimiento al meter el transportador
      SET;
      L     "DB602_ElementosQuimarox".Quimarox[#ID_Quimarox].Elementos[#ID_Elemento].Avance_carrier;  // #datos_elemento.Avance_carrier
      L     #Pto_Ajuste_6;
      >=I;
      JC    ErrorMoverPosicionReposo;  // error de movimiento al meter el transportador

/////////////////////////////////////////////////////////////////////////////////////
// Si ya no Ventana
      SET;
      AN    "DB602_ElementosQuimarox".Quimarox[#ID_Quimarox].Elementos[#ID_Elemento].Hay_Carrier_en_ventana;  // #datos_elemento.Hay_Carrier_en_ventana
      JC    ErrorMoverPosicionReposo;

      BE;

/////////////////////////////////////////////////////////////////////////////////////
ET08_VelocidadNormal:CLR;
      =     #ElevadorEnLenta;
      BE;

/////////////////////////////////////////////////////////////////////////////////////
ET08_IrEtapa_01_Vacia:CLR;
      =     #Ir_PosicionReposo;
      =     #Ir_PosicionCarga;
      =     #ElevadorEnLenta;

      L     1;
      T     #EstadoAsociadoEnMesa;
      BE;



NETWORK
TITLE = >>>>>>>>>>>>>>>>>>>>>>>>>>>>>>>>>>>>>>>>>>>>>>>>>>>>>>>>>>>>>>>>>>>

NETWORK
TITLE = ETAPA 10 >>> RESET CARGADO >>> Comprobar Ruta
/////////////////////////////////////////////////////////////////////////////////////
/////////////////////////////////////////////////////////////////////////////////////
// Extraer Destino
ETAPA_10_ResetCargado_ComprobarRuta:NOP   0;
      SET;
      =     "DB900_Estado_Mesas".EstadoVI[#MesaDeCarga].Etapas_Reset;


/////////////////////////////////////////////////////////////////////////////////////
      SET;
      =     #PararElevador;
      CLR;
      =     #Ir_PosicionCarga;
      =     #Ir_PosicionReposo;


/////////////////////////////////////////////////////////////////////////////////////
      SET;
      AN    #pHs_Protrusion;
      JC    ErrorProtrusion;


/////////////////////////////////////////////////////////////////////////////////////
/// --- Comprobacion del TIPO de MESA
      SET;
      AN    #EsMesaTL;
      JC    ET10_TRACKING_ComprobarRuta;
      JU    ET10_ROUTING_ComprobarRuta;


/////////////////////////////////////////////////////////////////////////////////////
/////////////////////////////////////////////////////////////////////////////////////
/////////////////////////////////////////////////////////////////////////////////////
/// --- Comprobacion de Ruta en una MESA de ROUTING
ET10_ROUTING_ComprobarRuta:NOP   0;
      L     #ROUTING_Destino;
      L     0;
      ==I;
      JC    ErrorDatosCargada;
      JU    ET10_FINAL_ComprobacionDeRuta;

/////////////////////////////////////////////////////////////////////////////////////
/////////////////////////////////////////////////////////////////////////////////////
/////////////////////////////////////////////////////////////////////////////////////
/// --- Comprobacion de Ruta en una MESA de TRACKING
ET10_TRACKING_ComprobarRuta:NOP   0;
      L     "DB810_ColasMesas".Colas[#MesaDeCarga].UT_PrimeraMesa;
      T     #NumeroUT;

      SET;
      L     #NumeroUT;  // Debe existir UT
      L     0;
      ==I;
      JC    ErrorDatosCargada;

// si la mesa actual es la de destino, es que aun no tiene ruta, y tenemos que esperar
      SET;
      L     "DB812_UTs_Control".UT[#NumeroUT].MesaActual;
      L     "DB812_UTs_Control".UT[#NumeroUT].MesaDestino;
      ==I;
      JC    ErrorDatosCargada;

      SET;
      L     0;
      L     "DB812_UTs_Control".UT[#NumeroUT].MesaDestino;
      ==I;
      JC    ErrorDatosCargada;

      JU    ET10_FINAL_ComprobacionDeRuta;

/////////////////////////////////////////////////////////////////////////////////////
/////////////////////////////////////////////////////////////////////////////////////
/////////////////////////////////////////////////////////////////////////////////////
/// --- Final de la Comprobacion de Ruta
//      si tenemos destino, esperamos aviso
ET10_FINAL_ComprobacionDeRuta:NOP   0;
      SET;
      A     #PRV_AVTF;
      JC    ET10_IrEtapa_07_FinCargaDelPeine;

      BE;

/////////////////////////////////////////////////////////////////////////////////////
ET10_IrEtapa_07_FinCargaDelPeine:NOP   0;
      L     7;
      T     #EstadoAsociadoEnMesa;
      JU    ETAPA_07_FinCargaDelPeine;



NETWORK
TITLE = ETAPA 11 >>> RESET VACIO >>> Mover Posicion de Reposo
/////////////////////////////////////////////////////////////////////////////////////
/////////////////////////////////////////////////////////////////////////////////////
/////////////////////////////////////////////////////////////////////////////////////
ETAPA_11_ResetVacio_MoverPosicionDeReposo:NOP   0;
      SET;
      =     "DB900_Estado_Mesas".EstadoVI[#MesaDeCarga].Etapas_Reset;


/////////////////////////////////////////////////////////////////////////////////////
      SET;
      A     #En_PosicionReposo;
      JC    ET11_IrEtapa_1_Reset_EnReposo;


/////////////////////////////////////////////////////////////////////////////////////
      SET;
      =     #Ir_PosicionReposo;
      =     #PararElevador;
      CLR;
      =     #Ir_PosicionCarga;

/////////////////////////////////////////////////////////////////////////////////////
      SET;
      AN    #pHs_Protrusion;
      JC    ErrorProtrusion;

      BE;


/////////////////////////////////////////////////////////////////////////////////////
/////////////////////////////////////////////////////////////////////////////////////
/////////////////////////////////////////////////////////////////////////////////////
ET11_IrEtapa_1_Reset_EnReposo:NOP   0;
      CLR;
      =     #Ir_PosicionReposo;
      =     #Ir_PosicionCarga;

      L     1;
      T     #EstadoAsociadoEnMesa;
      JU    ETAPA_01_EnReposo;


NETWORK
TITLE = >>>>>>>>>>>>>>>>>>>>>>>>>>>>>>>>>>>>>>>>>>>>>>>>>>>>>>>>>>>>>>>>>>>

NETWORK
TITLE = ERRRORES DE LA MESA >>> Activacion
/////////////////////////////////////////////////////////////////////////////////////
/////////////////////////////////////////////////////////////////////////////////////
/////////////////////////////////////////////////////////////////////////////////////
ErrorProtrusion:NOP   0;
      SET;
      =     "DB900_Estado_Mesas".EstadoVI[#MesaDeCarga].Error_Mx;
      =     "DB900_Estado_Mesas".EstadoVI[#MesaDeCarga].Err_Protusion;
      =     #PararElevador;
      BE;

/////////////////////////////////////////////////////////////////////////////////////
/////////////////////////////////////////////////////////////////////////////////////
/////////////////////////////////////////////////////////////////////////////////////
ErrorCargaDelPeine:NOP   0;  // error en la carga
      SET;
      =     "DB900_Estado_Mesas".EstadoVI[#MesaDeCarga].Err_TOut_Avance_E1_E3;
      =     "DB900_Estado_Mesas".EstadoVI[#MesaDeCarga].Error_Mx;
      =     #PararElevador;
      BE;

/////////////////////////////////////////////////////////////////////////////////////
/////////////////////////////////////////////////////////////////////////////////////
/////////////////////////////////////////////////////////////////////////////////////
ErrorMoverPosicionCarga:SET;
      =     #PararElevador;
      =     "DB900_Estado_Mesas".EstadoVI[#MesaDeCarga].Error_Mx;
      =     "DB900_Estado_Mesas".EstadoVI[#MesaDeCarga].Err_Tout_Sacar;
      BE;

/////////////////////////////////////////////////////////////////////////////////////
/////////////////////////////////////////////////////////////////////////////////////
/////////////////////////////////////////////////////////////////////////////////////
ErrorMoverPosicionReposo:SET;
      =     #PararElevador;
      =     "DB900_Estado_Mesas".EstadoVI[#MesaDeCarga].Error_Mx;
      =     "DB900_Estado_Mesas".EstadoVI[#MesaDeCarga].Err_Tout_Recoger;
      BE;

/////////////////////////////////////////////////////////////////////////////////////
/////////////////////////////////////////////////////////////////////////////////////
/////////////////////////////////////////////////////////////////////////////////////
ErrorDatosCargada:NOP   0;  // error en la carga
      SET;
      =     "DB900_Estado_Mesas".EstadoVI[#MesaDeCarga].Error_Mx;
      =     "DB900_Estado_Mesas".EstadoVI[#MesaDeCarga].Err_DatosPLC;
      =     #PararElevador;
      BE;



NETWORK
TITLE = FINAL DE LA FUNCION
/////////////////////////////////////////////////////////////////////////////////////
/////////////////////////////////////////////////////////////////////////////////////
/////////////////////////////////////////////////////////////////////////////////////
FinFuncion:BE;


END_FUNCTION_BLOCK
